SUBAPPLICATION Baumsetzer (* Hauptapplikation des ISOBUS-Baumsetzers: verknuepft Bedienelemente (Buttons/Softkeys), den Automatikablauf (Start_Baumsetzer), die Aktoren (Granulatschieber, Luftventil, Summer, Wasserpumpe, Wasserventil), den Baumzaehler sowie die Statusanzeigen (Hintergrundfarben, Scheinwerfer) auf dem Terminal *)
  (* Standard: 61499-2 *)
  (* Version 1.0, 2024-04-23, Elias *)
  PACKAGE FBs::Baumsetzer;
  IMPORT DataPanel::io::MI::DQ::DataPanel_MI_DO::DigitalOutput_6A;
  IMPORT DataPanel::io::MI::const::MI::MI_00;
  IMPORT isobus::UT::Q::const::colours::COLOR_GREEN;
  IMPORT isobus::UT::Q::const::colours::COLOR_RED;
  IMPORT isobus::UT::io::Button::ButtonActivationCode::BT_RELEASED_UNLATCHED;
  IMPORT isobus::UT::io::Softkey::SoftKeyActivationCode::SK_RELEASED;
  IMPORT test::FBs::Baumsetzer::Constants::DefaultPool::Button_Granulatschieber;
  IMPORT test::FBs::Baumsetzer::Constants::DefaultPool::Button_Luftventil;
  IMPORT test::FBs::Baumsetzer::Constants::DefaultPool::Button_Reset_Baeume_gepflanzt;
  IMPORT test::FBs::Baumsetzer::Constants::DefaultPool::Button_Summer;
  IMPORT test::FBs::Baumsetzer::Constants::DefaultPool::Button_Wasserpumpe;
  IMPORT test::FBs::Baumsetzer::Constants::DefaultPool::Button_Wasserventil;
  IMPORT test::FBs::Baumsetzer::Constants::DefaultPool::SoftKey_Scheinwerfer;
  IMPORT test::FBs::Baumsetzer::Constants::DefaultPool::Start;
  IMPORT test::FBs::Baumsetzer::Constants::DefaultPool::Stop;
  FBS
    OR_1 : iec61131::bitwiseOperators::OR_2(IN1 := BOOL#FALSE, IN2 := BOOL#FALSE, OUT := BOOL#FALSE {SET_ATTRIBUTE(Attribute1, )});
    SoftKey_F2 : isobus::UT::io::Softkey::Softkey_IE(QI := TRUE, u16ObjId := Stop, InputEvent := SK_RELEASED);
    F_AND : iec61131::bitwiseOperators::AND_2(IN1 := BOOL#FALSE, IN2 := BOOL#FALSE);
    F_AND_1 : iec61131::bitwiseOperators::AND_2;
    OR_2 : iec61131::bitwiseOperators::OR_2(IN1 := BOOL#FALSE, IN2 := BOOL#FALSE, OUT := BOOL#FALSE);
    F_AND_2 : iec61131::bitwiseOperators::AND_2;
    OR_3 : iec61131::bitwiseOperators::OR_2(IN1 := BOOL#FALSE, IN2 := BOOL#FALSE, OUT := BOOL#FALSE);
    F_AND_3 : iec61131::bitwiseOperators::AND_2;
    OR_4 : iec61131::bitwiseOperators::OR_2(IN1 := BOOL#FALSE, IN2 := BOOL#FALSE, OUT := BOOL#FALSE);
    OR_5 : iec61131::bitwiseOperators::OR_2(IN1 := BOOL#FALSE, IN2 := BOOL#FALSE, OUT := BOOL#FALSE);
    F_AND_4 : iec61131::bitwiseOperators::AND_2;
    E_SR : iec61499::events::E_SR;
    E_SWITCH : iec61499::events::E_SWITCH;
    Button_Granulatschieber : isobus::UT::io::Button::Button_IE(QI := TRUE, u16ObjId := Button_Granulatschieber, InputEvent := BT_RELEASED_UNLATCHED);
    Button_Luftventil : isobus::UT::io::Button::Button_IE(QI := TRUE, u16ObjId := Button_Luftventil, InputEvent := BT_RELEASED_UNLATCHED);
    Button_Summer : isobus::UT::io::Button::Button_IE(QI := TRUE, u16ObjId := Button_Summer, InputEvent := BT_RELEASED_UNLATCHED);
    Button_Wasserpumpe : isobus::UT::io::Button::Button_IE(QI := TRUE, u16ObjId := Button_Wasserpumpe, InputEvent := BT_RELEASED_UNLATCHED);
    Button_Wasserventil : isobus::UT::io::Button::Button_IE(QI := TRUE, u16ObjId := Button_Wasserventil, InputEvent := BT_RELEASED_UNLATCHED);
    E_PULSE : iec61499::events::timers::E_PULSE(PT := T#120s);
    E_PULSE_1 : iec61499::events::timers::E_PULSE(PT := T#120s);
    E_PULSE_2 : iec61499::events::timers::E_PULSE(PT := T#120s);
    E_PULSE_3 : iec61499::events::timers::E_PULSE(PT := T#120s);
    E_PULSE_4 : iec61499::events::timers::E_PULSE(PT := T#120s);
    E_PERMIT : iec61499::events::E_PERMIT;
    Q_BackgroundColour : isobus::UT::Q::Q_BackgroundColour(u16ObjId := Button_Luftventil);
    F_SEL : iec61131::selection::F_SEL(IN0 := COLOR_RED, IN1 := COLOR_GREEN);
    F_SEL_1 : iec61131::selection::F_SEL(IN0 := COLOR_RED, IN1 := COLOR_GREEN);
    Q_BackgroundColour_1 : isobus::UT::Q::Q_BackgroundColour(u16ObjId := Button_Granulatschieber);
    F_SEL_2 : iec61131::selection::F_SEL(IN0 := COLOR_RED, IN1 := COLOR_GREEN);
    Q_BackgroundColour_2 : isobus::UT::Q::Q_BackgroundColour(u16ObjId := Button_Summer);
    F_SEL_3 : iec61131::selection::F_SEL(IN0 := COLOR_RED, IN1 := COLOR_GREEN);
    Q_BackgroundColour_3 : isobus::UT::Q::Q_BackgroundColour(u16ObjId := Button_Wasserpumpe);
    F_SEL_4 : iec61131::selection::F_SEL(IN0 := COLOR_RED, IN1 := COLOR_GREEN);
    Q_BackgroundColour_4 : isobus::UT::Q::Q_BackgroundColour(u16ObjId := Button_Wasserventil);
    SoftKey_F6 : isobus::UT::io::Softkey::Softkey_IX(QI := TRUE, PARAMS := '', u16ObjId := SoftKey_Scheinwerfer);
    Scheinwerfer : DataPanel::io::MI::DQ::DataPanel_MI_QX(QI := TRUE, u8SAMember := MI_00, Output := DigitalOutput_6A);
    Q_BackgroundColour_5 : isobus::UT::Q::Q_BackgroundColour(u16ObjId := Start);
    F_SEL_5 : iec61131::selection::F_SEL(IN0 := COLOR_RED, IN1 := COLOR_GREEN);
    Q_BackgroundColour_6 : isobus::UT::Q::Q_BackgroundColour(u16ObjId := Stop);
    F_SEL_6 : iec61131::selection::F_SEL(IN0 := COLOR_RED, IN1 := COLOR_GREEN);
    F_NOT : iec61131::bitwiseOperators::F_NOT;
    Button_Reset_Baeume_gepflanzt : isobus::UT::io::Button::Button_IE(QI := TRUE, u16ObjId := Button_Reset_Baeume_gepflanzt, InputEvent := BT_RELEASED_UNLATCHED);
    F_BOOL_TO_DWORD : iec61131::conversion::F_BOOL_TO_DWORD;
    F_BOOL_TO_DWORD_1 : iec61131::conversion::F_BOOL_TO_DWORD;
    F_BOOL_TO_DWORD_2 : iec61131::conversion::F_BOOL_TO_DWORD;
    F_BOOL_TO_DWORD_3 : iec61131::conversion::F_BOOL_TO_DWORD;
    F_BOOL_TO_DWORD_4 : iec61131::conversion::F_BOOL_TO_DWORD;
    E_T_FF : iec61499::events::E_T_FF;
    Q_BackgroundColour_7 : isobus::UT::Q::Q_BackgroundColour(u16ObjId := Button_Luftventil);
    F_SEL_7 : iec61131::selection::F_SEL(IN0 := COLOR_RED, IN1 := COLOR_GREEN);
  END_FBS
  SUBAPPS
    Luftventil : Luftventil;
    Summer : Summer;
    Wasserpumpe : Wasserpumpe;
    Wasserventil : Wasserventil;
    Start_Baumsetzer : FBs::Baumsetzer::func::Automatik::Start_Baumsetzer;
    Baumzaehler : FBs::Baumsetzer::func::Zaehlermenue::Baumzaehler;
    Granulatschieber : Granulatschieber;
  END_SUBAPPS
  EVENT_CONNECTIONS
    F_AND_1.CNF TO Luftventil.REQ;
    F_AND_2.CNF TO Summer.REQ;
    F_AND_3.CNF TO Wasserpumpe.REQ;
    F_AND_4.CNF TO Wasserventil.REQ;
    E_SR.EO TO F_AND.REQ;
    E_SR.EO TO F_AND_1.REQ;
    E_SR.EO TO F_AND_2.REQ;
    E_SR.EO TO F_AND_4.REQ;
    E_SR.EO TO F_AND_3.REQ;
    SoftKey_F2.IND TO E_SR.R;
    F_AND.CNF TO Granulatschieber.REQ;
    SoftKey_F2.IND TO Start_Baumsetzer.STOP;
    Start_Baumsetzer.Start TO E_SR.S;
    Summer.CNF TO E_SWITCH.EI;
    Start_Baumsetzer.Pulse_Wasser TO OR_5.REQ;
    Start_Baumsetzer.Pulse_Wasserpumpe TO OR_4.REQ;
    Start_Baumsetzer.Pulse_Summer TO OR_3.REQ;
    Start_Baumsetzer.Pulse_Luft TO OR_2.REQ;
    Start_Baumsetzer.Pulse_Granulat TO OR_1.REQ;
    Button_Granulatschieber.IND TO E_PULSE.REQ;
    E_PULSE.CNF TO OR_1.REQ;
    Button_Luftventil.IND TO E_PULSE_1.REQ;
    Button_Summer.IND TO E_PULSE_2.REQ;
    Button_Wasserpumpe.IND TO E_PULSE_3.REQ;
    Button_Wasserventil.IND TO E_PULSE_4.REQ;
    E_PULSE_1.CNF TO OR_2.REQ;
    E_PULSE_2.CNF TO OR_3.REQ;
    E_PULSE_3.CNF TO OR_4.REQ;
    E_PULSE_4.CNF TO OR_5.REQ;
    Button_Granulatschieber.IND TO E_SR.S;
    Button_Luftventil.IND TO E_SR.S;
    Button_Summer.IND TO E_SR.S;
    Button_Wasserpumpe.IND TO E_SR.S;
    Button_Wasserventil.IND TO E_SR.S;
    E_SWITCH.EO1 TO E_PERMIT.EI;
    E_PERMIT.EO TO Baumzaehler.CU;
    F_SEL.CNF TO Q_BackgroundColour.REQ;
    F_AND_1.CNF TO F_SEL.REQ;
    F_SEL_1.CNF TO Q_BackgroundColour_1.REQ;
    F_AND.CNF TO F_SEL_1.REQ;
    F_SEL_2.CNF TO Q_BackgroundColour_2.REQ;
    F_AND_2.CNF TO F_SEL_2.REQ;
    F_SEL_3.CNF TO Q_BackgroundColour_3.REQ;
    F_AND_3.CNF TO F_SEL_3.REQ;
    F_SEL_4.CNF TO Q_BackgroundColour_4.REQ;
    F_AND_4.CNF TO F_SEL_4.REQ;
    SoftKey_F2.IND TO E_PULSE.R;
    SoftKey_F2.IND TO E_PULSE_1.R;
    SoftKey_F2.IND TO E_PULSE_2.R;
    SoftKey_F2.IND TO E_PULSE_3.R;
    SoftKey_F2.IND TO E_PULSE_4.R;
    SoftKey_F6.IND TO E_T_FF.CLK;
    F_SEL_5.CNF TO Q_BackgroundColour_5.REQ;
    E_SR.EO TO F_SEL_5.REQ;
    E_SR.EO TO F_NOT.REQ;
    F_SEL_6.CNF TO Q_BackgroundColour_6.REQ;
    F_NOT.CNF TO F_SEL_6.REQ;
    F_BOOL_TO_DWORD.CNF TO F_AND.REQ;
    F_BOOL_TO_DWORD_1.CNF TO F_AND_1.REQ;
    F_BOOL_TO_DWORD_2.CNF TO F_AND_2.REQ;
    F_BOOL_TO_DWORD_3.CNF TO F_AND_3.REQ;
    F_BOOL_TO_DWORD_4.CNF TO F_AND_4.REQ;
    Button_Reset_Baeume_gepflanzt.IND TO Baumzaehler.RESET;
    OR_1.CNF TO F_BOOL_TO_DWORD.REQ;
    OR_2.CNF TO F_BOOL_TO_DWORD_1.REQ;
    OR_3.CNF TO F_BOOL_TO_DWORD_2.REQ;
    OR_4.CNF TO F_BOOL_TO_DWORD_3.REQ;
    OR_5.CNF TO F_BOOL_TO_DWORD_4.REQ;
    E_T_FF.EO TO Scheinwerfer.REQ;
    E_T_FF.EO TO F_SEL_7.REQ;
    F_SEL_7.CNF TO Q_BackgroundColour_7.REQ;
  END_CONNECTIONS
  DATA_CONNECTIONS
    F_AND_1.OUT TO Luftventil.OUT;
    F_AND_2.OUT TO Summer.OUT;
    F_AND_3.OUT TO Wasserpumpe.OUT;
    F_AND_4.OUT TO Wasserventil.OUT;
    E_SR.Q TO F_AND.IN2;
    E_SR.Q TO F_AND_1.IN2;
    E_SR.Q TO F_AND_2.IN2;
    E_SR.Q TO F_AND_3.IN2;
    E_SR.Q TO F_AND_4.IN2;
    F_AND.OUT TO Granulatschieber.OUT;
    F_AND_2.OUT TO E_SWITCH.G;
    Start_Baumsetzer.Wasserventil TO OR_5.IN1;
    Start_Baumsetzer.Wasserpumpe TO OR_4.IN1;
    Start_Baumsetzer.Summer TO OR_3.IN1;
    Start_Baumsetzer.Luftventil TO OR_2.IN1;
    Start_Baumsetzer.Granulatschieber TO OR_1.IN1;
    E_PULSE.Q TO OR_1.IN2;
    E_PULSE_1.Q TO OR_2.IN2;
    E_PULSE_2.Q TO OR_3.IN2;
    E_PULSE_3.Q TO OR_4.IN2;
    E_PULSE_4.Q TO OR_5.IN2;
    Start_Baumsetzer.Summer TO E_PERMIT.PERMIT;
    F_SEL.OUT TO Q_BackgroundColour.u8Colour;
    F_AND_1.OUT TO F_SEL.G;
    F_SEL_1.OUT TO Q_BackgroundColour_1.u8Colour;
    F_AND.OUT TO F_SEL_1.G;
    F_SEL_2.OUT TO Q_BackgroundColour_2.u8Colour;
    F_AND_2.OUT TO F_SEL_2.G;
    F_SEL_3.OUT TO Q_BackgroundColour_3.u8Colour;
    F_AND_3.OUT TO F_SEL_3.G;
    F_SEL_4.OUT TO Q_BackgroundColour_4.u8Colour;
    F_AND_4.OUT TO F_SEL_4.G;
    F_SEL_5.OUT TO Q_BackgroundColour_5.u8Colour;
    E_SR.Q TO F_SEL_5.G;
    E_SR.Q TO F_NOT.IN;
    F_SEL_6.OUT TO Q_BackgroundColour_6.u8Colour;
    F_NOT.OUT TO F_SEL_6.G;
    F_BOOL_TO_DWORD.OUT TO F_AND.IN1;
    F_BOOL_TO_DWORD_1.OUT TO F_AND_1.IN1;
    F_BOOL_TO_DWORD_2.OUT TO F_AND_2.IN1;
    F_BOOL_TO_DWORD_3.OUT TO F_AND_3.IN1;
    F_BOOL_TO_DWORD_4.OUT TO F_AND_4.IN1;
    OR_1.OUT TO F_BOOL_TO_DWORD.IN;
    OR_2.OUT TO F_BOOL_TO_DWORD_1.IN;
    OR_3.OUT TO F_BOOL_TO_DWORD_2.IN;
    OR_4.OUT TO F_BOOL_TO_DWORD_3.IN;
    OR_5.OUT TO F_BOOL_TO_DWORD_4.IN;
    E_T_FF.Q TO Scheinwerfer.OUT;
    E_T_FF.Q TO F_SEL_7.G;
    F_SEL_7.OUT TO Q_BackgroundColour_7.u8Colour;
  END_CONNECTIONS
END_SUBAPPLICATION
